// TIA Portal V17 export
// export: Created 2024-08-29T18:23:47.5788601Z, ExportSetting WithDefaults, DisplayName Totally Integrated Automation Portal, DisplayVersion V17 Update 7, DisplayName TIA Portal Openness, DisplayVersion V17 Update 7, DisplayName TIA Portal Version Control Interface, DisplayVersion V17, DisplayName SINAMICS Startdrive Advanced, DisplayVersion V17 SP2, DisplayName SINAMICS Startdrive G110M, G120, G120C, G120D, G120P, G115D, DisplayVersion V17 SP2, DisplayName SINAMICS Startdrive G130, G150, S120, S150, SINAMICS MV, S210, DisplayVersion V17 SP2, DisplayName STEP 7 Professional, DisplayVersion V17 Update 7, DisplayName STEP 7 Safety, DisplayVersion V17 Update 6, DisplayName WinCC Advanced / Unified PC, DisplayVersion V17 Update 7
FUNCTION_BLOCK "FC_IJCORE_MAIN"   // FB1000, LAD
{ S7_Optimized_Access := 'FALSE' }
VERSION : 0.1
// stored: AutoNumber false, IsIECCheckEnabled false, SetENOAutomatically false, UDAEnableTagReadback false
   VAR DB_SPECIFIC
      Enable : Bool;
      Mode : Int;
      Indicator : Int;
      AlarmReset : Bool;
      NFP : Array[1..5] of String[30];
   END_VAR
   VAR
      AWK : "FB_IJC_AWAKE_SIGNAL";
      MSG : Array[1..20] of "FB_IJC_PROTOCOL";
   END_VAR
   VAR DB_SPECIFIC
      Faults : Array[0..1] of Word;
   END_VAR
   VAR
      FaultsArray AT Faults : Array[1..32] of Bool;
   END_VAR
   VAR_TEMP
      "return" : Bool;
      i : Int;
      ERROR_STR : String;
   END_VAR
BEGIN

REGION Network 1: Fault Reset
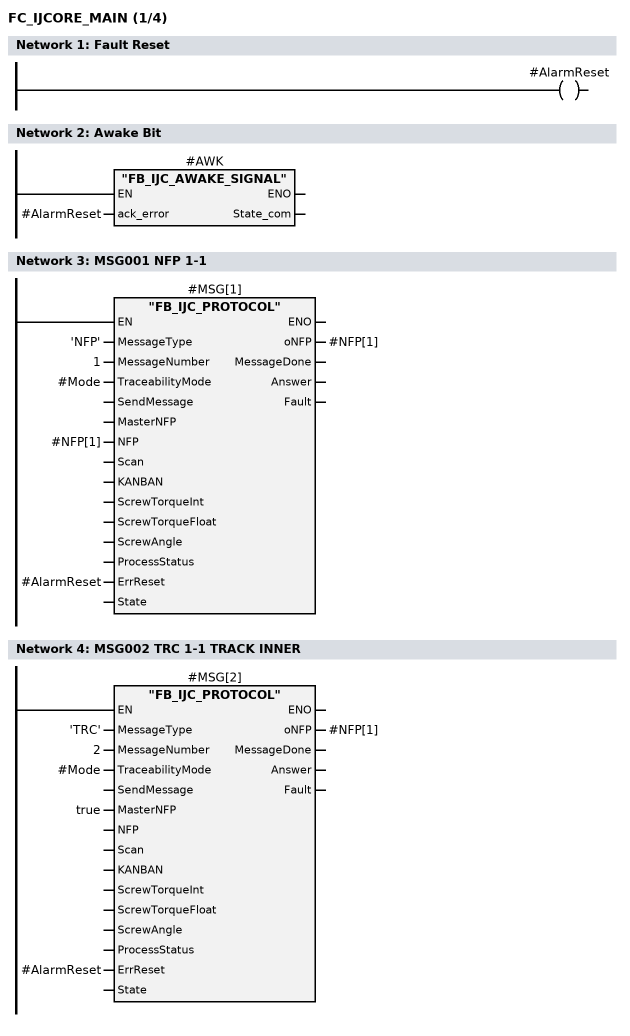
   RUNG wire#powerrail
      Coil( #AlarmReset )
   END_RUNG
   // the same network as SCL:
   #AlarmReset := TRUE;
END_REGION

REGION Network 2: Awake Bit
   RUNG wire#powerrail
      #AWK(ack_error := #AlarmReset, State_com =>)
   END_RUNG
   // the same network as SCL:
   #AWK(ack_error := #AlarmReset);   // "FB_IJC_AWAKE_SIGNAL"
END_REGION

REGION Network 3: MSG001 NFP 1-1
   RUNG wire#powerrail
      #MSG[1](MessageType := 'NFP', MessageNumber := 1, TraceabilityMode := #Mode, SendMessage :=, MasterNFP :=, NFP := #NFP[1], Scan :=, KANBAN :=, ScrewTorqueInt :=, ScrewTorqueFloat :=, ScrewAngle :=, ProcessStatus :=, ErrReset := #AlarmReset, State :=, oNFP => #NFP[1], MessageDone =>, Answer =>, Fault =>)
   END_RUNG
   // the same network as SCL:
   #MSG[1](MessageType := 'NFP',   // "FB_IJC_PROTOCOL"
           MessageNumber := 1,
           TraceabilityMode := #Mode,
           NFP := #NFP[1],
           ErrReset := #AlarmReset,
           oNFP => #NFP[1]);
END_REGION

REGION Network 4: MSG002 TRC 1-1 TRACK INNER
   RUNG wire#powerrail
      #MSG[2](MessageType := 'TRC', MessageNumber := 2, TraceabilityMode := #Mode, SendMessage :=, MasterNFP := true, NFP :=, Scan :=, KANBAN :=, ScrewTorqueInt :=, ScrewTorqueFloat :=, ScrewAngle :=, ProcessStatus :=, ErrReset := #AlarmReset, State :=, oNFP => #NFP[1], MessageDone =>, Answer =>, Fault =>)
   END_RUNG
   // the same network as SCL:
   #MSG[2](MessageType := 'TRC',   // "FB_IJC_PROTOCOL"
           MessageNumber := 2,
           TraceabilityMode := #Mode,
           MasterNFP := true,
           ErrReset := #AlarmReset,
           oNFP => #NFP[1]);
END_REGION

REGION Network 5: MSG003 TRC 1-2 TRACK OUTER
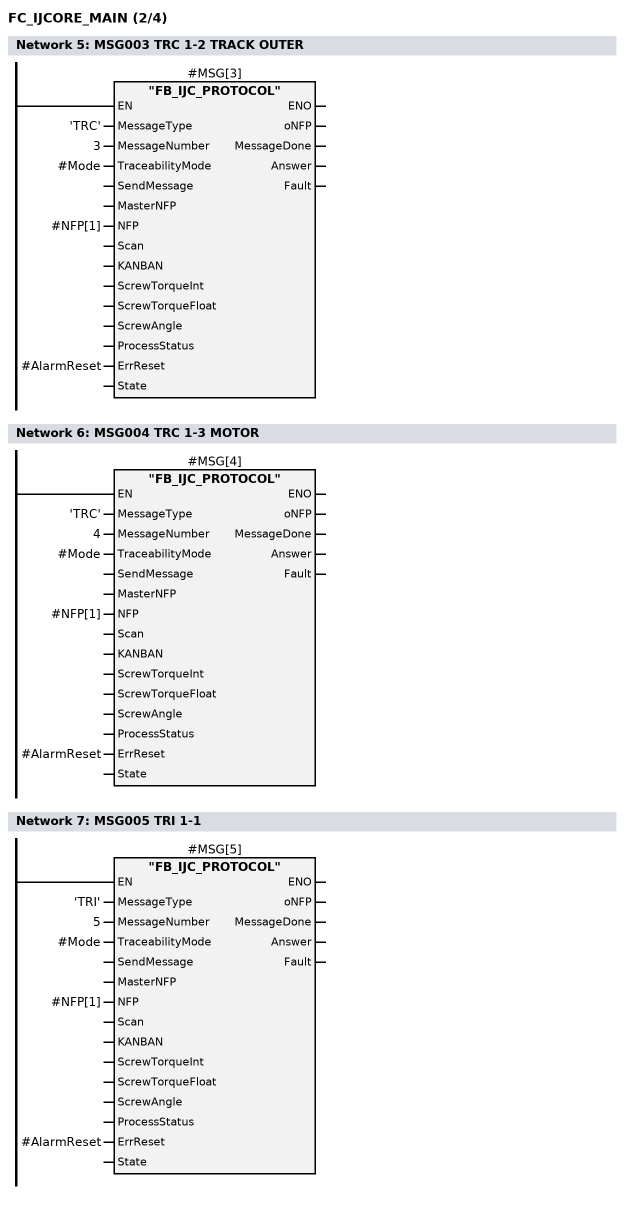
   RUNG wire#powerrail
      #MSG[3](MessageType := 'TRC', MessageNumber := 3, TraceabilityMode := #Mode, SendMessage :=, MasterNFP :=, NFP := #NFP[1], Scan :=, KANBAN :=, ScrewTorqueInt :=, ScrewTorqueFloat :=, ScrewAngle :=, ProcessStatus :=, ErrReset := #AlarmReset, State :=, oNFP =>, MessageDone =>, Answer =>, Fault =>)
   END_RUNG
   // the same network as SCL:
   #MSG[3](MessageType := 'TRC',   // "FB_IJC_PROTOCOL"
           MessageNumber := 3,
           TraceabilityMode := #Mode,
           NFP := #NFP[1],
           ErrReset := #AlarmReset);
END_REGION

REGION Network 6: MSG004 TRC 1-3 MOTOR
   RUNG wire#powerrail
      #MSG[4](MessageType := 'TRC', MessageNumber := 4, TraceabilityMode := #Mode, SendMessage :=, MasterNFP :=, NFP := #NFP[1], Scan :=, KANBAN :=, ScrewTorqueInt :=, ScrewTorqueFloat :=, ScrewAngle :=, ProcessStatus :=, ErrReset := #AlarmReset, State :=, oNFP =>, MessageDone =>, Answer =>, Fault =>)
   END_RUNG
   // the same network as SCL:
   #MSG[4](MessageType := 'TRC',   // "FB_IJC_PROTOCOL"
           MessageNumber := 4,
           TraceabilityMode := #Mode,
           NFP := #NFP[1],
           ErrReset := #AlarmReset);
END_REGION

REGION Network 7: MSG005 TRI 1-1
   RUNG wire#powerrail
      #MSG[5](MessageType := 'TRI', MessageNumber := 5, TraceabilityMode := #Mode, SendMessage :=, MasterNFP :=, NFP := #NFP[1], Scan :=, KANBAN :=, ScrewTorqueInt :=, ScrewTorqueFloat :=, ScrewAngle :=, ProcessStatus :=, ErrReset := #AlarmReset, State :=, oNFP =>, MessageDone =>, Answer =>, Fault =>)
   END_RUNG
   // the same network as SCL:
   #MSG[5](MessageType := 'TRI',   // "FB_IJC_PROTOCOL"
           MessageNumber := 5,
           TraceabilityMode := #Mode,
           NFP := #NFP[1],
           ErrReset := #AlarmReset);
END_REGION

REGION Network 8: MSG006 CNF 1-1 TRACK INNER
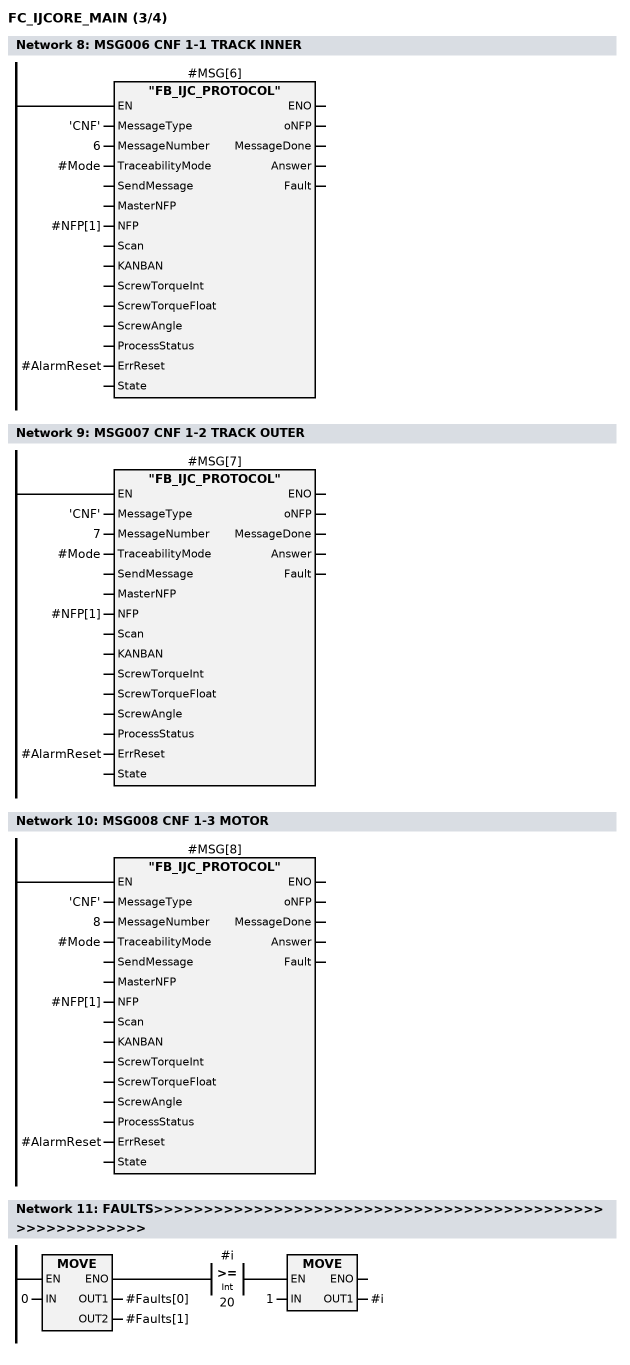
   RUNG wire#powerrail
      #MSG[6](MessageType := 'CNF', MessageNumber := 6, TraceabilityMode := #Mode, SendMessage :=, MasterNFP :=, NFP := #NFP[1], Scan :=, KANBAN :=, ScrewTorqueInt :=, ScrewTorqueFloat :=, ScrewAngle :=, ProcessStatus :=, ErrReset := #AlarmReset, State :=, oNFP =>, MessageDone =>, Answer =>, Fault =>)
   END_RUNG
   // the same network as SCL:
   #MSG[6](MessageType := 'CNF',   // "FB_IJC_PROTOCOL"
           MessageNumber := 6,
           TraceabilityMode := #Mode,
           NFP := #NFP[1],
           ErrReset := #AlarmReset);
END_REGION

REGION Network 9: MSG007 CNF 1-2 TRACK OUTER
   RUNG wire#powerrail
      #MSG[7](MessageType := 'CNF', MessageNumber := 7, TraceabilityMode := #Mode, SendMessage :=, MasterNFP :=, NFP := #NFP[1], Scan :=, KANBAN :=, ScrewTorqueInt :=, ScrewTorqueFloat :=, ScrewAngle :=, ProcessStatus :=, ErrReset := #AlarmReset, State :=, oNFP =>, MessageDone =>, Answer =>, Fault =>)
   END_RUNG
   // the same network as SCL:
   #MSG[7](MessageType := 'CNF',   // "FB_IJC_PROTOCOL"
           MessageNumber := 7,
           TraceabilityMode := #Mode,
           NFP := #NFP[1],
           ErrReset := #AlarmReset);
END_REGION

REGION Network 10: MSG008 CNF 1-3 MOTOR
   RUNG wire#powerrail
      #MSG[8](MessageType := 'CNF', MessageNumber := 8, TraceabilityMode := #Mode, SendMessage :=, MasterNFP :=, NFP := #NFP[1], Scan :=, KANBAN :=, ScrewTorqueInt :=, ScrewTorqueFloat :=, ScrewAngle :=, ProcessStatus :=, ErrReset := #AlarmReset, State :=, oNFP =>, MessageDone =>, Answer =>, Fault =>)
   END_RUNG
   // the same network as SCL:
   #MSG[8](MessageType := 'CNF',   // "FB_IJC_PROTOCOL"
           MessageNumber := 8,
           TraceabilityMode := #Mode,
           NFP := #NFP[1],
           ErrReset := #AlarmReset);
END_REGION

REGION Network 11: FAULTS>>>>>>>>>>>>>>>>>>>>>>>>>>>>>>>>>>>>>>>>>>>>>>>>>>>>>>>>>>
   RUNG wire#powerrail
      Move(in := 0, out1 => #Faults[0], out2 => #Faults[1])
      { S7_Templates := "SrcType := Int" } GE_Contact(in1 := #i, in2 := 20)
      Move(in := 1, out1 => #i)
   END_RUNG
   // the same network as SCL:
   #Faults[0] := 0;
   #Faults[1] := 0;
   IF #i >= 20 THEN #i := 1; END_IF;
END_REGION

REGION Network 12: Awake bit
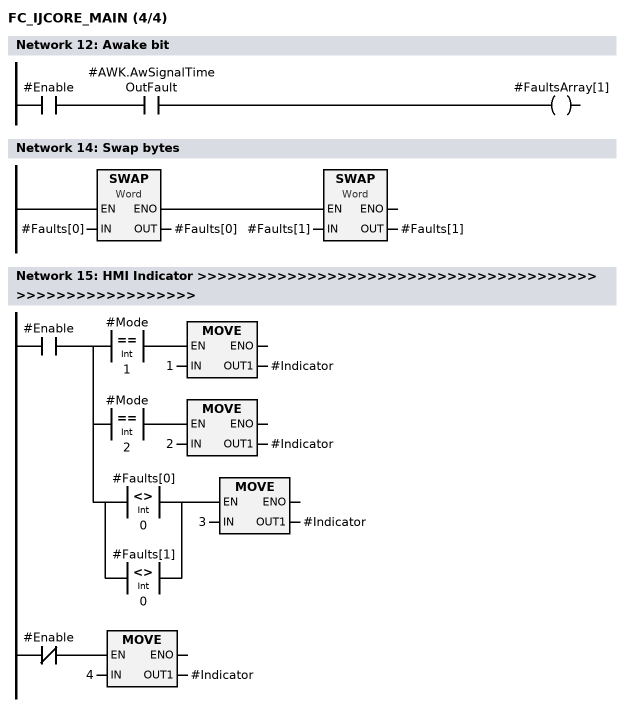
   RUNG wire#powerrail
      Contact( #Enable )
      Contact( #AWK.AwSignalTimeOutFault )
      Coil( #FaultsArray[1] )
   END_RUNG
   // the same network as SCL:
   #FaultsArray[1] := #Enable AND #AWK.AwSignalTimeOutFault;
END_REGION

REGION Network 13 (SCL): Answer faults
   FOR #i := 1 TO 20 DO
       CASE #MSG[#i].Answer OF
           -2:  // NFP not founded
               #FaultsArray[2] := TRUE;
           -3:  //Part number NOT inside BOM
               #FaultsArray[3] := TRUE;
           -4: // PFC not ok
               #FaultsArray[4] := TRUE;
           -5: //Component already used
               #FaultsArray[5] := true;
           -6: //Module already used
               #FaultsArray[6] := true;
           -10: //Status NOK from previous operation
               #FaultsArray[10] := true;

       END_CASE;



   END_FOR;
END_REGION

REGION Network 14: Swap bytes
   #Faults[0] := SWAP(#Faults[0]);
   #Faults[1] := SWAP(#Faults[1]);
END_REGION

REGION Network 15: HMI Indicator >>>>>>>>>>>>>>>>>>>>>>>>>>>>>>>>>>>>>>>>>>>>>>>>>>>>>>>>>>
   RUNG wire#powerrail
      Contact( #Enable )
      wire#w1
      { S7_Templates := "SrcType := Int" } EQ_Contact(in1 := #Mode, in2 := 1)
      Move(in := 1, out1 => #Indicator)
   END_RUNG
   RUNG wire#w1
      { S7_Templates := "SrcType := Int" } EQ_Contact(in1 := #Mode, in2 := 2)
      Move(in := 2, out1 => #Indicator)
   END_RUNG
   RUNG wire#w1
      { S7_Templates := "SrcType := Int" } NE_Contact(in1 := #Faults[0], in2 := 0)
      wire#w2
      Move(in := 3, out1 => #Indicator)
   END_RUNG
   RUNG wire#w1
      { S7_Templates := "SrcType := Int" } NE_Contact(in1 := #Faults[1], in2 := 0)
   END_RUNG wire#w2
   RUNG wire#powerrail
      I_Contact( #Enable )
      Move(in := 4, out1 => #Indicator)
   END_RUNG
   // the same network as SCL:
   IF #Enable AND (#Mode = 1) THEN #Indicator := 1; END_IF;
   IF #Enable AND (#Mode = 2) THEN #Indicator := 2; END_IF;
   IF #Enable AND ((#Faults[0] <> 0) OR (#Faults[1] <> 0)) THEN #Indicator := 3; END_IF;
   IF NOT #Enable THEN #Indicator := 4; END_IF;
END_REGION
END_FUNCTION_BLOCK
